TYPE FsT_ErrMsg : STRING(FsParam_ErrorHandling.ERROR_MSG_SIZE); END_TYPE

(* stored: Version 1.1.0.1, ProductVersion 3.1.4024.4
   DUT FsT_ErrMsg: Id {6c14e48e-c2e0-4815-af44-424aae3b6f77} *)
